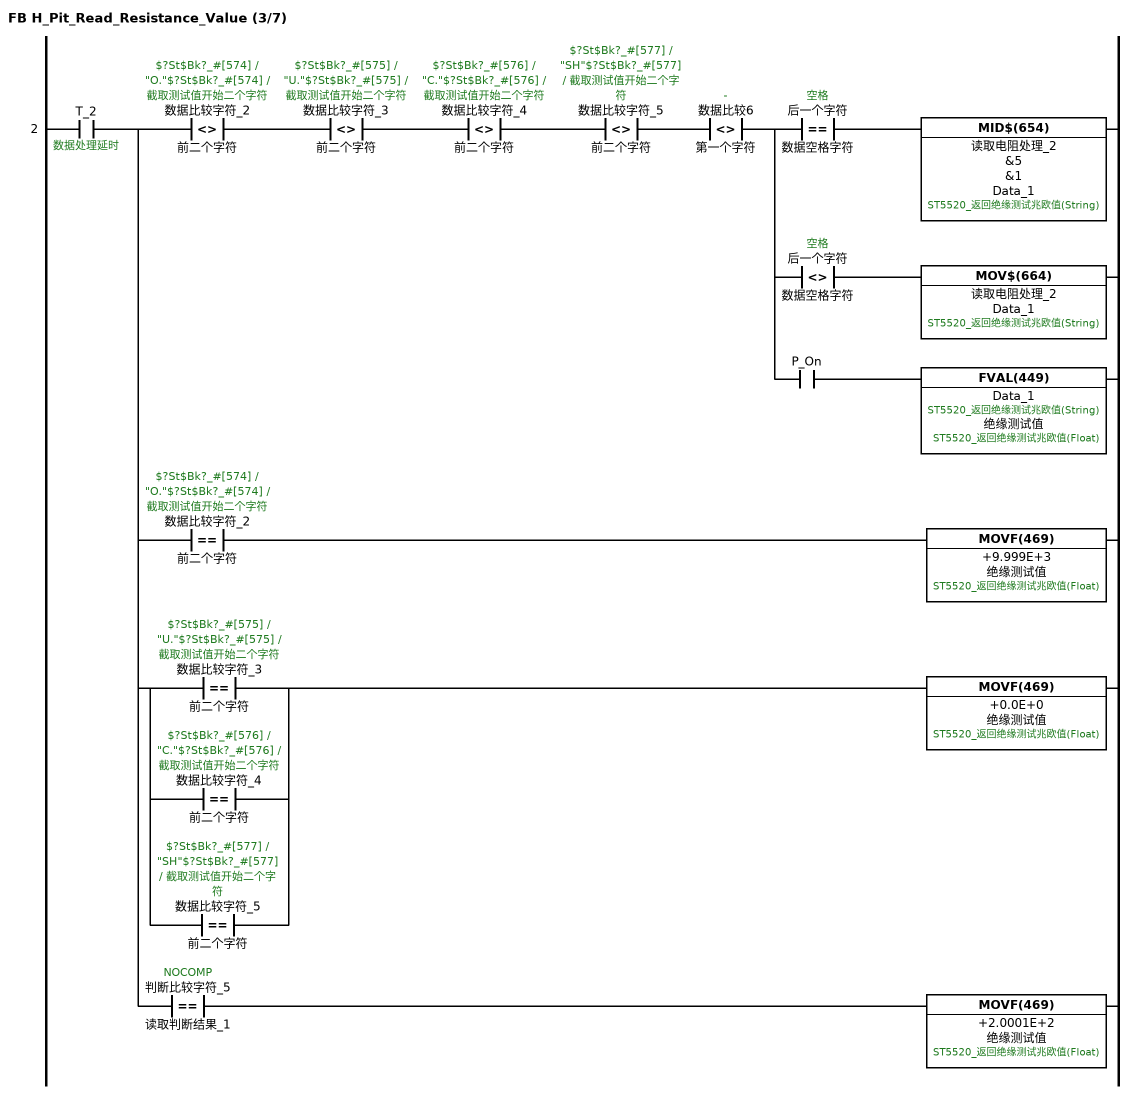
; [picture p264: FB H_Pit_Read_Resistance_Value, rungs 2-2]
; rung 2
LD T_2  ; 数据处理延时
OUT TR0
AND<>(305) 数据比较字符_2 前二个字符  ; $?St$Bk?_#[574] / "O."$?St$Bk?_#[574], 截取测试值开始二个字符
AND<>(305) 数据比较字符_3 前二个字符  ; $?St$Bk?_#[575] / "U."$?St$Bk?_#[575], 截取测试值开始二个字符
AND<>(305) 数据比较字符_4 前二个字符  ; $?St$Bk?_#[576] / "C."$?St$Bk?_#[576], 截取测试值开始二个字符
AND<>(305) 数据比较字符_5 前二个字符  ; $?St$Bk?_#[577] / "SH"$?St$Bk?_#[577], 截取测试值开始二个字符
AND<>(305) 数据比较6 第一个字符  ; -
OUT TR1
AND=(300) 后一个字符 数据空格字符  ; 空格
MID$(654) 读取电阻处理_2 &5 &1 Data_1  ; ST5520_返回绝缘测试兆欧值(String)
LD TR1
AND<>(305) 后一个字符 数据空格字符  ; 空格
MOV$(664) 读取电阻处理_2 Data_1  ; ST5520_返回绝缘测试兆欧值(String)
LD TR1
AND P_On
FVAL(449) Data_1 绝缘测试值  ; ST5520_返回绝缘测试兆欧值(String), ST5520_返回绝缘测试兆欧值(Float)
LD TR0
AND=(300) 数据比较字符_2 前二个字符  ; $?St$Bk?_#[574] / "O."$?St$Bk?_#[574], 截取测试值开始二个字符
MOVF(469) +9.999E+3 绝缘测试值  ; ST5520_返回绝缘测试兆欧值(Float)
LD TR0
LD=(300) 数据比较字符_3 前二个字符  ; $?St$Bk?_#[575] / "U."$?St$Bk?_#[575], 截取测试值开始二个字符
OR=(300) 数据比较字符_4 前二个字符  ; $?St$Bk?_#[576] / "C."$?St$Bk?_#[576], 截取测试值开始二个字符
OR=(300) 数据比较字符_5 前二个字符  ; $?St$Bk?_#[577] / "SH"$?St$Bk?_#[577], 截取测试值开始二个字符
ANDLD
MOVF(469) +0.0E+0 绝缘测试值  ; ST5520_返回绝缘测试兆欧值(Float)
LD TR0
AND=(300) 判断比较字符_5 读取判断结果_1  ; NOCOMP
MOVF(469) +2.0001E+2 绝缘测试值  ; ST5520_返回绝缘测试兆欧值(Float)

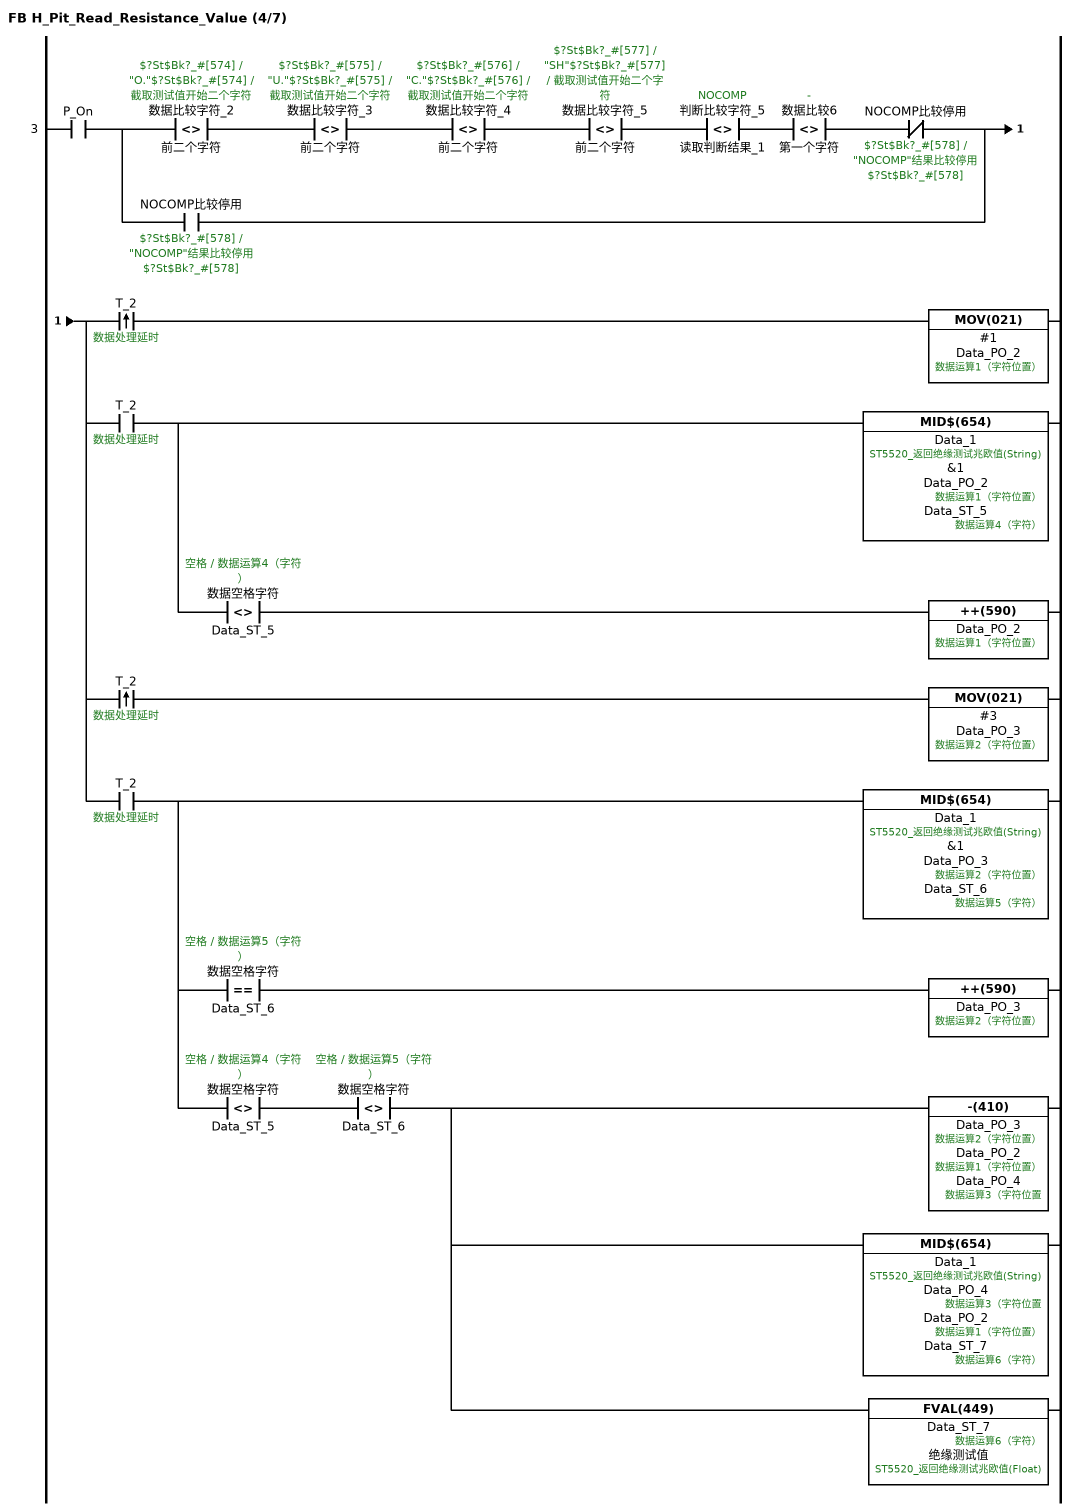
; rung 3
LD P_On
LD<>(305) 数据比较字符_2 前二个字符  ; $?St$Bk?_#[574] / "O."$?St$Bk?_#[574], 截取测试值开始二个字符
AND<>(305) 数据比较字符_3 前二个字符  ; $?St$Bk?_#[575] / "U."$?St$Bk?_#[575], 截取测试值开始二个字符
AND<>(305) 数据比较字符_4 前二个字符  ; $?St$Bk?_#[576] / "C."$?St$Bk?_#[576], 截取测试值开始二个字符
AND<>(305) 数据比较字符_5 前二个字符  ; $?St$Bk?_#[577] / "SH"$?St$Bk?_#[577], 截取测试值开始二个字符
AND<>(305) 判断比较字符_5 读取判断结果_1  ; NOCOMP
AND<>(305) 数据比较6 第一个字符  ; -
ANDNOT NOCOMP比较停用  ; $?St$Bk?_#[578] / "NOCOMP"结果比较停用$?St$Bk?_#[578]
OR NOCOMP比较停用  ; $?St$Bk?_#[578] / "NOCOMP"结果比较停用$?St$Bk?_#[578]
ANDLD
OUT TR0
@AND T_2  ; 数据处理延时
MOV(021) #1 Data_PO_2  ; 数据运算1（字符位置）
LD TR0
AND T_2  ; 数据处理延时
MID$(654) Data_1 &1 Data_PO_2 Data_ST_5  ; ST5520_返回绝缘测试兆欧值(String), 数据运算1（字符位置）, 数据运算4（字符）
AND<>(305) 数据空格字符 Data_ST_5  ; 空格, 数据运算4（字符）
++(590) Data_PO_2  ; 数据运算1（字符位置）
LD TR0
@AND T_2  ; 数据处理延时
MOV(021) #3 Data_PO_3  ; 数据运算2（字符位置）
LD TR0
AND T_2  ; 数据处理延时
OUT TR1
MID$(654) Data_1 &1 Data_PO_3 Data_ST_6  ; ST5520_返回绝缘测试兆欧值(String), 数据运算2（字符位置）, 数据运算5（字符）
AND=(300) 数据空格字符 Data_ST_6  ; 空格, 数据运算5（字符）
++(590) Data_PO_3  ; 数据运算2（字符位置）
LD TR1
AND<>(305) 数据空格字符 Data_ST_5  ; 空格, 数据运算4（字符）
AND<>(305) 数据空格字符 Data_ST_6  ; 空格, 数据运算5（字符）
-(410) Data_PO_3 Data_PO_2 Data_PO_4  ; 数据运算2（字符位置）, 数据运算1（字符位置）, 数据运算3（字符位置
MID$(654) Data_1 Data_PO_4 Data_PO_2 Data_ST_7  ; ST5520_返回绝缘测试兆欧值(String), 数据运算3（字符位置, 数据运算1（字符位置）, 数据运算6（字符）
FVAL(449) Data_ST_7 绝缘测试值  ; 数据运算6（字符）, ST5520_返回绝缘测试兆欧值(Float)

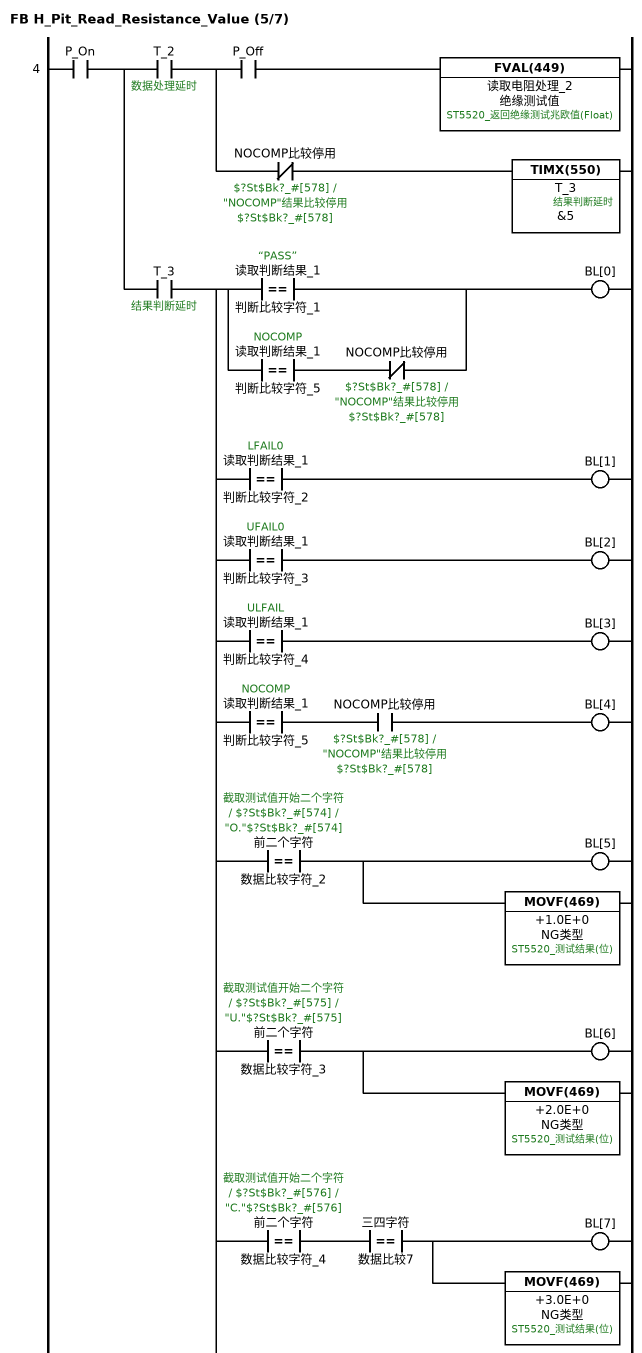

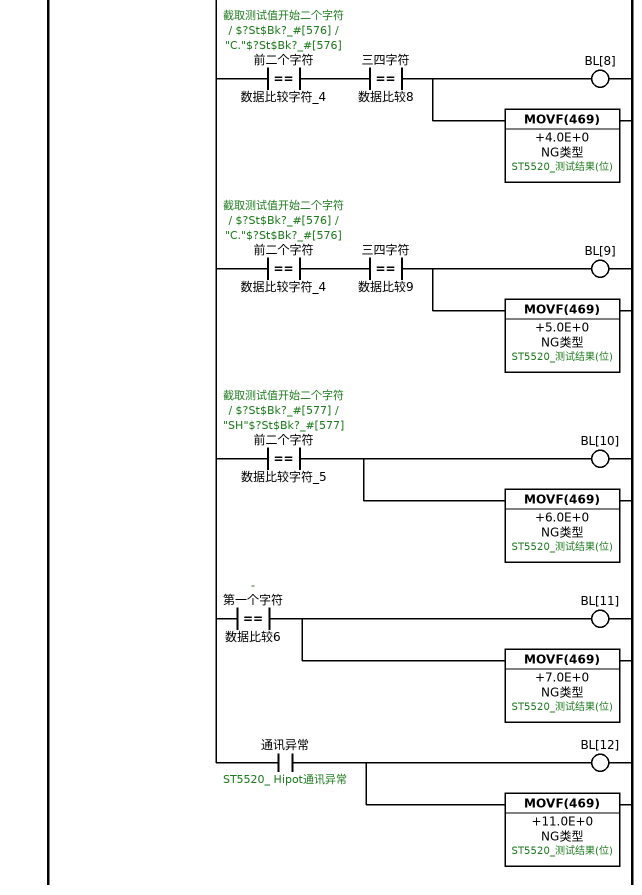
; rung 4
LD P_On
OUT TR0
AND T_2  ; 数据处理延时
OUT TR1
AND P_Off
FVAL(449) 读取电阻处理_2 绝缘测试值  ; ST5520_返回绝缘测试兆欧值(Float)
LD TR1
ANDNOT NOCOMP比较停用  ; $?St$Bk?_#[578] / "NOCOMP"结果比较停用$?St$Bk?_#[578]
TIMX(550) T_3 &5  ; 结果判断延时
LD TR0
AND T_3  ; 结果判断延时
OUT TR2
LD=(300) 读取判断结果_1 判断比较字符_1  ; “PASS”
LD=(300) 读取判断结果_1 判断比较字符_5  ; NOCOMP
ANDNOT NOCOMP比较停用  ; $?St$Bk?_#[578] / "NOCOMP"结果比较停用$?St$Bk?_#[578]
ORLD
ANDLD
OUT BL[0]
LD TR2
AND=(300) 读取判断结果_1 判断比较字符_2  ; LFAIL0
OUT BL[1]
LD TR2
AND=(300) 读取判断结果_1 判断比较字符_3  ; UFAIL0
OUT BL[2]
LD TR2
AND=(300) 读取判断结果_1 判断比较字符_4  ; ULFAIL
OUT BL[3]
LD TR2
AND=(300) 读取判断结果_1 判断比较字符_5  ; NOCOMP
AND NOCOMP比较停用  ; $?St$Bk?_#[578] / "NOCOMP"结果比较停用$?St$Bk?_#[578]
OUT BL[4]
LD TR2
AND=(300) 前二个字符 数据比较字符_2  ; 截取测试值开始二个字符, $?St$Bk?_#[574] / "O."$?St$Bk?_#[574]
OUT BL[5]
MOVF(469) +1.0E+0 NG类型  ; ST5520_测试结果(位)
LD TR2
AND=(300) 前二个字符 数据比较字符_3  ; 截取测试值开始二个字符, $?St$Bk?_#[575] / "U."$?St$Bk?_#[575]
OUT BL[6]
MOVF(469) +2.0E+0 NG类型  ; ST5520_测试结果(位)
LD TR2
AND=(300) 前二个字符 数据比较字符_4  ; 截取测试值开始二个字符, $?St$Bk?_#[576] / "C."$?St$Bk?_#[576]
AND=(300) 三四字符 数据比较7
OUT BL[7]
MOVF(469) +3.0E+0 NG类型  ; ST5520_测试结果(位)
LD TR2
AND=(300) 前二个字符 数据比较字符_4  ; 截取测试值开始二个字符, $?St$Bk?_#[576] / "C."$?St$Bk?_#[576]
AND=(300) 三四字符 数据比较8
OUT BL[8]
MOVF(469) +4.0E+0 NG类型  ; ST5520_测试结果(位)
LD TR2
AND=(300) 前二个字符 数据比较字符_4  ; 截取测试值开始二个字符, $?St$Bk?_#[576] / "C."$?St$Bk?_#[576]
AND=(300) 三四字符 数据比较9
OUT BL[9]
MOVF(469) +5.0E+0 NG类型  ; ST5520_测试结果(位)
LD TR2
AND=(300) 前二个字符 数据比较字符_5  ; 截取测试值开始二个字符, $?St$Bk?_#[577] / "SH"$?St$Bk?_#[577]
OUT BL[10]
MOVF(469) +6.0E+0 NG类型  ; ST5520_测试结果(位)
LD TR2
AND=(300) 第一个字符 数据比较6  ; -
OUT BL[11]
MOVF(469) +7.0E+0 NG类型  ; ST5520_测试结果(位)
LD TR2
AND 通讯异常  ; ST5520_ Hipot通讯异常
OUT BL[12]
MOVF(469) +11.0E+0 NG类型  ; ST5520_测试结果(位)

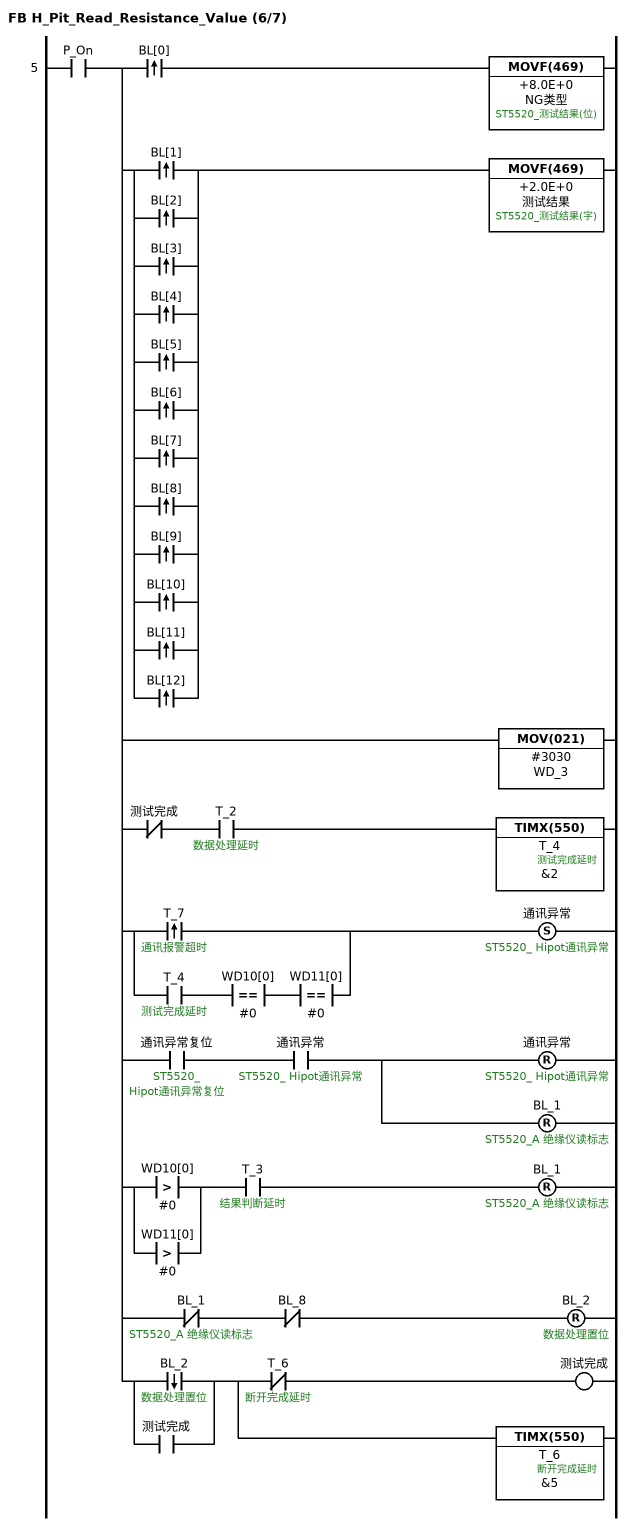
; rung 5
LD P_On
OUT TR0
@AND BL[0]
MOVF(469) +8.0E+0 NG类型  ; ST5520_测试结果(位)
LD TR0
@LD BL[1]
@OR BL[2]
@OR BL[3]
@OR BL[4]
@OR BL[5]
@OR BL[6]
@OR BL[7]
@OR BL[8]
@OR BL[9]
@OR BL[10]
@OR BL[11]
@OR BL[12]
ANDLD
MOVF(469) +2.0E+0 测试结果  ; ST5520_测试结果(字)
LD TR0
MOV(021) #3030 WD_3
ANDNOT 测试完成
AND T_2  ; 数据处理延时
TIMX(550) T_4 &2  ; 测试完成延时
LD TR0
@LD T_7  ; 通讯报警超时
LD T_4  ; 测试完成延时
AND=(300) WD10[0] #0
AND=(300) WD11[0] #0
ORLD
ANDLD
SET 通讯异常  ; ST5520_ Hipot通讯异常
LD TR0
AND 通讯异常复位  ; ST5520_Hipot通讯异常复位
AND 通讯异常  ; ST5520_ Hipot通讯异常
RSET 通讯异常  ; ST5520_ Hipot通讯异常
RSET BL_1  ; ST5520_A 绝缘仪读标志
LD TR0
LD>(320) WD10[0] #0
OR>(320) WD11[0] #0
ANDLD
AND T_3  ; 结果判断延时
RSET BL_1  ; ST5520_A 绝缘仪读标志
LD TR0
ANDNOT BL_1  ; ST5520_A 绝缘仪读标志
ANDNOT BL_8
RSET BL_2  ; 数据处理置位
LD TR0
%LD BL_2  ; 数据处理置位
OR 测试完成
ANDLD
OUT TR1
ANDNOT T_6  ; 断开完成延时
OUT 测试完成
LD TR1
TIMX(550) T_6 &5  ; 断开完成延时

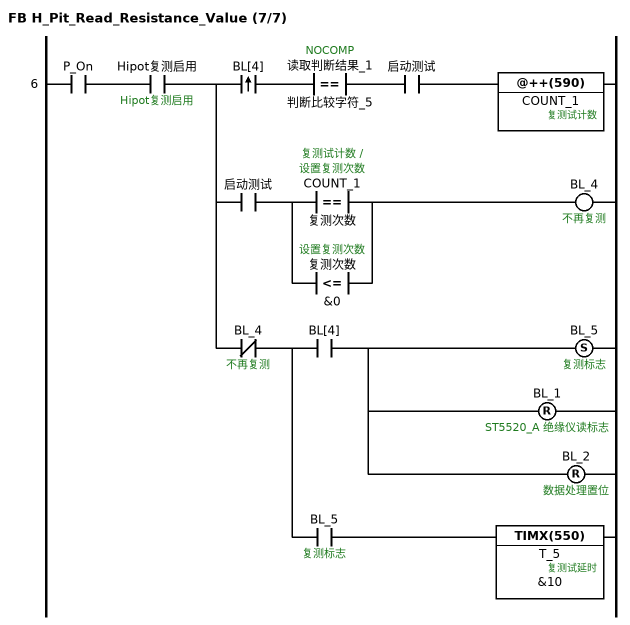
; rung 6
LD P_On
AND Hipot复测启用  ; Hipot复测启用
OUT TR0
@AND BL[4]
AND=(300) 读取判断结果_1 判断比较字符_5  ; NOCOMP
AND 启动测试
@++(590) COUNT_1  ; 复测试计数
LD TR0
AND 启动测试
LD=(300) COUNT_1 复测次数  ; 复测试计数, 设置复测次数
OR<=(315) 复测次数 &0  ; 设置复测次数
ANDLD
OUT BL_4  ; 不再复测
LD TR0
ANDNOT BL_4  ; 不再复测
OUT TR1
AND BL[4]
SET BL_5  ; 复测标志
RSET BL_1  ; ST5520_A 绝缘仪读标志
RSET BL_2  ; 数据处理置位
LD TR1
AND BL_5  ; 复测标志
TIMX(550) T_5 &10  ; 复测试延时

## Function block P_change
VAR_INPUT
  P_IN : INT;  (* 压力输入 *)
  P_B : REAL := 1.0;  (* 压力倍率 *)
  P_C : REAL;  (* 补偿值 *)
END_VAR
VAR_OUTPUT
  P_OUT : DINT;  (* 转换后的压力 *)
END_VAR
VAR
  P_F : REAL;  (* 压力值—浮点 *)
  P_ADV : REAL;  (* 压力值—倍率后 *)
  P_ADD : REAL;  (* 压力值—补偿后 *)
  NC : BOOL := TRUE;
END_VAR

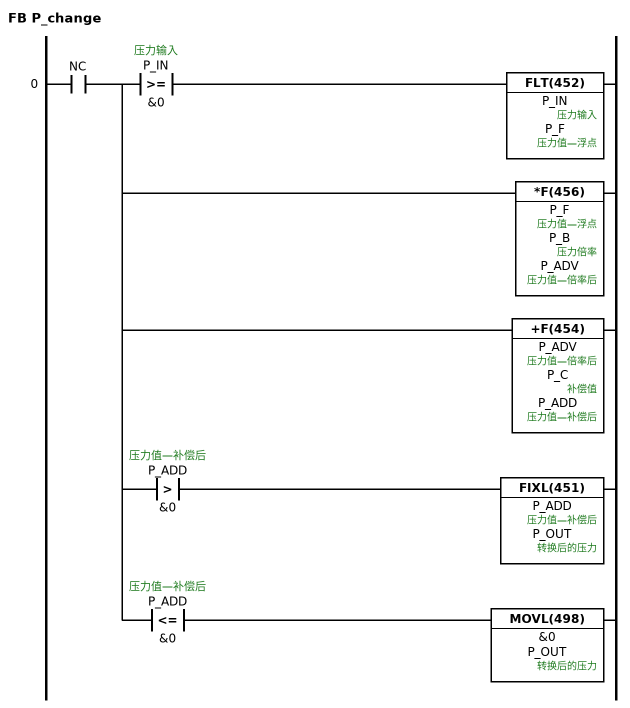
; rung 0
LD NC
OUT TR0
AND>=(325) P_IN &0  ; 压力输入
FLT(452) P_IN P_F  ; 压力输入, 压力值—浮点
LD TR0
*F(456) P_F P_B P_ADV  ; 压力值—浮点, 压力倍率, 压力值—倍率后
+F(454) P_ADV P_C P_ADD  ; 压力值—倍率后, 补偿值, 压力值—补偿后
AND>F(333) P_ADD &0  ; 压力值—补偿后
FIXL(451) P_ADD P_OUT  ; 压力值—补偿后, 转换后的压力
LD TR0
AND<=F(332) P_ADD &0  ; 压力值—补偿后
MOVL(498) &0 P_OUT  ; 转换后的压力